(* CODESYS project ELEVADOR.project

Project tree, tasks and I/O mapping:
  Device : CODESYS Control Win V3, 3S - Smart Software Solutions GmbH, order no. 305021, version 3.5.11.30
    application Application
      libraries: Standard, * (System)
      task MainTask (cyclic, interval t#20ms, priority 1) calls PLC_PRG
      program PLC_PRG [LD]
*)

// Device/Application/PLC_PRG
PROGRAM PLC_PRG
VAR
	BT1F : BOOL;          // BOTAO DE PESSAO EXETRIOR PRIMEIRO ANDAR
    BT2F : BOOL;          // BOTAO DE PESSAO EXETRIOR SEGUNDO ANDAR
    BT1D : BOOL;          // BOTAO DE PESSAO INTERIOR PRIMERIO ANDAR
    BT2D : BOOL;          // BOTAO DE PESSAO INTERIOR SEGUNDO ANDAR
    LBT1 : BOOL;          // LUZ DO BOTAO 1 EXTERIOR
    LBT2 : BOOL;          // LUZ DO BOTAO 2 EXTERIOR
    F2 : BOOL;            // FIM DE CURSO PISO SUPERIOR
    F1 : BOOL;            // FIM DE CURSO PISO INFERIOR
    FPA : BOOL;           // FIM DE CURSO PORTA ABERTA
    FPF : BOOL;           // FIM DE CURSO PORTA FECHADA
    SS  : BOOL;           // SENSOR DE SEGURANÇA ALGUEM NO CAMINHO DA PORTA
	P1: BOOL;
	P2: BOOL;
END_VAR

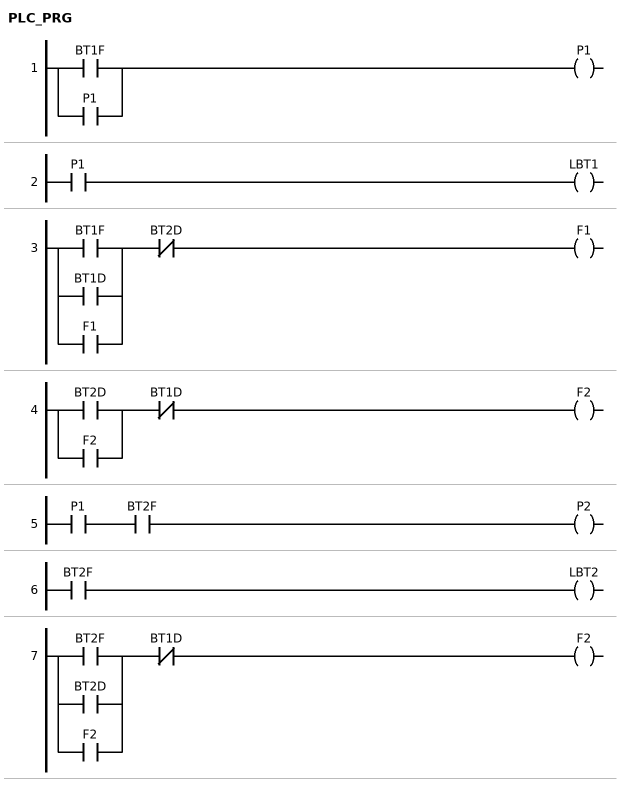
// NETWORK 1
P1 := BT1F OR P1;

// NETWORK 2
LBT1 := P1;

// NETWORK 3
F1 := (BT1F OR BT1D OR F1) AND NOT BT2D;

// NETWORK 4
F2 := (BT2D OR F2) AND NOT BT1D;

// NETWORK 5
P2 := P1 AND BT2F;

// NETWORK 6
LBT2 := BT2F;

// NETWORK 7
F2 := (BT2F OR BT2D OR F2) AND NOT BT1D;

END_PROGRAM
